VAR_GLOBAL CONSTANT

	cOversamples:DINT:=101;

END_VAR
VAR_GLOBAL

END_VAR

(* stored: Version 1.1.0.1
   GVL GVL: Id {9f9fa5d3-dcd2-43f0-9f7e-4d9c91afe4eb} *)
